(*
Nazwa:			FB_ReasonBadPackage
Opis:			Powód odrzuceń 
Wersja:			v0.1
Data:			2019-12-17
Autor:			DP
Urzadzenia:		
Konfiguracja:	
Info: 
- 
*)
FUNCTION_BLOCK FB_ReasonBadPackage
VAR_INPUT
	bEnable: BOOL;				//Zezwolenie na pracę
	bReset:BOOL;				//Stop awaryjny nieaktywny
	tTime:TIME;					//
	bAddReason:BOOL;			//Dodaj pomiar
	bReason1:BOOL;
	sReason1Description:STRING;	//Nazwa stacji nr 1
	bReason2:BOOL;
	sReason2Description:STRING;	//Nazwa stacji nr 2
	bReason3:BOOL;
	sReason3Description:STRING;	//Nazwa stacji nr 3
	bReason4:BOOL;
	sReason4Description:STRING;	//Nazwa stacji nr 4
	bReason5:BOOL;
	sReason5Description:STRING;	//Nazwa stacji nr 5
	bReason6:BOOL;
	sReason6Description:STRING;	//Nazwa stacji nr 6
	bReason7:BOOL;
	sReason7Description:STRING;	//Nazwa stacji nr 7
	bReason8:BOOL;
	sReason8Description:STRING;	//Nazwa stacji nr 8
	bReason9:BOOL;
	sReason9Description:STRING;	//Nazwa stacji nr 9
	bReason10:BOOL;
	sReason10Description:STRING;	//Nazwa stacji nr 10
	bReason11:BOOL;
	sReason11Description:STRING;	//Nazwa stacji nr 10
	bReason12:BOOL;
	sReason12Description:STRING;	//Nazwa stacji nr 10
END_VAR

VAR_OUTPUT
	sBadPackage1:STRING;		//Opis powodu odrzuceń nr 1
	sBadPackage2:STRING;		//Opis powodu odrzuceń nr 2
	sBadPackage3:STRING;		//Opis powodu odrzuceń nr 3
	iBadPackage1:INT;			//Ilość dla powodu odrzuceń nr 1
	iBadPackage2:INT;			//Ilość dla powodu odrzuceń nr 2
	iBadPackage3:INT;			//Ilość dla powodu odrzuceń nr3
END_VAR

VAR
	arReason: ARRAY [1..12] OF S_CycleTimes;
	i: INT;
	rtAddReason: R_TRIG;
	tonResetCounters: TON;
	dTimeTempReason1: DINT;
	dTimeTempReason2: DINT;
	dTimeTempReason3: DINT;
END_VAR

ErrorHandling();
Cycle();
ManualMovements();
Statistics();

ACTION Cycle:
tonResetCounters(IN:=NOT tonResetCounters.Q, PT:=tTime); // Resetowanie liczników
tonResetCounters.ET;
IF tonResetCounters.Q THEN
	FOR i:=1 TO 12 DO
		arReason[i].dTime :=0;
	END_FOR
	sBadPackage1 := '';
	sBadPackage2 := '';
	sBadPackage3 := '';	
	iBadPackage1 := 0;
	iBadPackage2 := 0;
	iBadPackage3 := 0;	
END_IF

rtAddReason(CLK:=bAddReason,Q=>);
IF rtAddReason.Q THEN
	IF bReason1 THEN
		arReason[1].dTime := arReason[1].dTime +1 ;
	ELSIF bReason2 THEN		                
		arReason[2].dTime := arReason[2].dTime +1 ;
	ELSIF bReason3 THEN		                
		arReason[3].dTime := arReason[3].dTime +1 ;
	ELSIF bReason4 THEN		                
		arReason[4].dTime := arReason[4].dTime +1 ;
	ELSIF bReason5 THEN		                
		arReason[5].dTime := arReason[5].dTime +1 ;
	ELSIF bReason6 THEN		                
		arReason[6].dTime := arReason[6].dTime +1 ;
	ELSIF bReason7 THEN		                
		arReason[7].dTime := arReason[7].dTime +1 ;
	ELSIF bReason8 THEN		                
		arReason[8].dTime := arReason[8].dTime +1 ;
	ELSIF bReason9 THEN		                
		arReason[9].dTime := arReason[9].dTime +1 ;
	ELSIF bReason10 THEN		                
		arReason[10].dTime := arReason[10].dTime +1 ;
	ELSIF bReason11 THEN		                
		arReason[11].dTime := arReason[11].dTime +1 ;
	ELSIF bReason12 THEN		                
		arReason[12].dTime := arReason[12].dTime +1 ;
	END_IF
END_IF

dTimeTempReason1:=0;
dTimeTempReason2:=0;
dTimeTempReason3:=0;
arReason[1].bName:=sReason1Description;
arReason[2].bName:=sReason2Description;
arReason[3].bName:=sReason3Description;
arReason[4].bName:=sReason4Description;
arReason[5].bName:=sReason5Description;
arReason[6].bName:=sReason6Description;
arReason[7].bName:=sReason7Description;
arReason[8].bName:=sReason8Description;
arReason[9].bName:=sReason9Description;
arReason[10].bName:=sReason10Description;
arReason[11].bName:=sReason11Description;
arReason[12].bName:=sReason12Description;

IF rtAddReason.Q THEN

	FOR i:=1 TO 12 DO
		IF arReason[i].dTime > dTimeTempReason1 AND arReason[i].dTime > 0 THEN
			dTimeTempReason1:=arReason[i].dTime;
			//sBadPackage1:=CONCAT(arReason[i].bName,CONCAT(' : ',DINT_TO_STRING(dTimeTempReason1))); 
			sBadPackage1:=arReason[i].bName;
			iBadPackage1:=DINT_TO_INT(dTimeTempReason1);
		END_IF
	END_FOR
	
	FOR i:=1 TO 12 DO
		IF NOT (dTimeTempReason1 = arReason[i].dTime) AND arReason[i].dTime > 0 AND arReason[i].dTime > dTimeTempReason2 THEN
			dTimeTempReason2:=arReason[i].dTime;
			//sBadPackage2:=CONCAT(arReason[i].bName,CONCAT(' : ',DINT_TO_STRING(dTimeTempReason2))); 
			sBadPackage2:=arReason[i].bName;
			iBadPackage2:=DINT_TO_INT(dTimeTempReason2);
		END_IF
	END_FOR
		
	
	FOR i:=1 TO 12 DO
		IF NOT (dTimeTempReason1 = arReason[i].dTime) AND NOT (dTimeTempReason2 = arReason[i].dTime) AND arReason[i].dTime > 0 AND arReason[i].dTime > dTimeTempReason3 THEN
			dTimeTempReason3:=arReason[i].dTime;
			//sBadPackage3:=CONCAT(arReason[i].bName,CONCAT(' : ',DINT_TO_STRING(dTimeTempReason3))); 
			sBadPackage3:=arReason[i].bName;
			iBadPackage3:=DINT_TO_INT(dTimeTempReason3);
		END_IF
	END_FOR

END_IF
END_ACTION

ACTION ErrorHandling:

END_ACTION

ACTION ManualMovements:

END_ACTION

ACTION Statistics:

END_ACTION

END_FUNCTION_BLOCK

(* stored: Version 1.1.0.1, ProductVersion 3.1.4026.13, FileIdentifier f821e4c9fa92b65123c5b5a8b96bb357d571fdac, FileSignature 66ee3a2cba180e0755bebfad92299a7f1b98f70d5f4e5fcc38dade54e5d1219834d17a801364c7d9427fb9c5d9b06b00baa2cb2c91a9147c5d8678a6a3ec7c272c0085550a2a79f781ff3bf7fd00fdc69d6a85ae68ab662de6a5fba1bf6f06088dd5d91340fab852d705084a9c7d45b0d485af99f788e7468afea8b732d8f02ab86418795cf481d6fb311848e723310e68e6f62f8bffc4d3983ff33911b6705eabe9c0ecd900fdff8a03da0ba1c1d559fbc20f151798523848cb2ea5f0b56665c15396b2e1ace1afb983d94e3e47069963c19748e630d4ef0e295de0e804a2c171911964497c2818236f735d0939e5cbb902e2f889e24f9c2e62be264d1a2e83
   POU FB_ReasonBadPackage: Id {ab9044d8-7ba6-411e-859f-6c590f740321}, SpecialFunc None
   Action Cycle: Id {66ff47de-74dd-4514-98b7-544ce218b048}
   Action ErrorHandling: Id {1f159861-3139-48a2-b8f4-e3e8459d5429}
   Action ManualMovements: Id {4d1ea5ec-6b83-46b0-9a59-5210da57e406}
   Action Statistics: Id {7c2082e2-d689-4215-9d04-46f61896639c} *)
